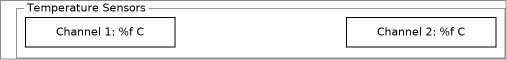
VISUALIZATION VISU_RTDs_4022  // 507x60
VAR_IN_OUT
	fTemp1 : LREAL;
	fTemp2 : LREAL;
END_VAR
    GroupBox (16,0 489x58), "Temperature Sensors"
        Rectangle (9,17 150x30), "Channel 1: %f C", text variable: fTemp1
            OnMouseDown: write the text variable via Default
        Rectangle (330,17 150x30), "Channel 2: %f C", tooltip "0 = Default Deceleration", text variable: fTemp2
            OnMouseDown: write the text variable via Default
END_VISUALIZATION

(* stored: Version 1.1.0.1, ProductVersion 3.1.4022.18
   Visu VISU_RTDs_4022: Id {d0831d85-ae1e-40f6-809a-db2dc438180f} *)
